# EPICS autosave request: iocBoot/iocTC32/auto_settings.req
file "TC32_settings.req", P=$(P)
